INTERFACE I_CH_List_Dublicate EXTENDS __SYSTEM.IQueryInterface

{attribute 'monitoring':='call'}
PROPERTY Content : REFERENCE TO ARRAY [1..BaseParameterlist.MAX_OBJECTS] OF I_CH_Object
GET
END_GET
END_PROPERTY

END_INTERFACE

(* stored: Version 1.1.0.1, ProductVersion 3.1.4024.13
   Itf I_CH_List_Dublicate: Id {dd5319f2-3bd5-4136-b363-8610e687c588}
   Property Content: Id {bc1cbc98-b44d-4fbc-baec-882d8bbbe01c}
   Get Get: Id {e8d98e35-cce7-4d8a-9eb2-34e8e7243909} *)
